TYPE ST_ProductionChange :
STRUCT
	MESSAGEHEADER  				: ST_MESSAGEHEADER;
	PRODUCTINFORMATION 			: ST_PRODUCTINFORMATION;
	PRODUCT						: ST_PRODUCT;
END_STRUCT
END_TYPE

(* stored: Version 1.1.0.1, ProductVersion 3.1.4024.13
   DUT ST_ProductionChange: Id {d28446c1-8f38-4b2f-981e-b8a6a383c685} *)
